// TIA Portal V17 export
// export: Created 2025-03-07T09:18:31.7382739Z, ExportSetting WithDefaults, DisplayName Totally Integrated Automation Portal, DisplayVersion V17 Update 8, DisplayName TIA Portal Openness, DisplayVersion V17 Update 8, DisplayName TIA Portal Version Control Interface, DisplayVersion V17, DisplayName SINAMICS Startdrive Advanced, DisplayVersion V17 SP2, DisplayName SINAMICS Startdrive G110M, G120, G120C, G120D, G120P, G115D, DisplayVersion V17 SP2, DisplayName SINAMICS Startdrive G130, G150, S120, S150, SINAMICS MV, S210, DisplayVersion V17 SP2, DisplayName STEP 7 Professional, DisplayVersion V17 Update 8, DisplayName SINUMERIK ONE STEP 7 Toolbox, DisplayVersion V17 Update 12, DisplayName SINUMERIK 840D sl STEP 7 Toolbox, DisplayVersion V17 Update 12, DisplayName STEP 7 Safety, DisplayVersion V17 Update 6, DisplayName WinCC Advanced, DisplayVersion V17 Update 8
DATA_BLOCK "LTLP_OperatingModeData"   // DB547
{ S7_Optimized_Access := 'FALSE'; DB_Accessible_From_OPC_UA := 'FALSE' }
VERSION : 0.1
// stored: AutoNumber true, DBAccessibleFromOPCUA false, DBAccessibleFromWebserver true, InstanceOfName LTLP_typeOperatingMode, InstanceOfType UDT, IsOnlyStoredInLoadMemory false, IsWriteProtectedInAS false
"LTLP_typeOperatingMode"
   // VAR RETAIN
   //    automaticMode : Struct
   //       tlFunctionAutomaticMode { S7_SetPoint := 'True'} : "LTLP_typeEnableFucntions";
   //       tlFunctionSingleMode { S7_SetPoint := 'True'} : "LTLP_typeEnableFucntions";
   //       tlFunctionSingleStepMode { S7_SetPoint := 'True'} : "LTLP_typeEnableFucntions";
   //       tlFunctionSetupMode { S7_SetPoint := 'True'} : "LTLP_typeEnableFucntions";
   //    END_STRUCT;
   //    setupMode : Struct
   //       tlFunctionSetupMode { S7_SetPoint := 'True'} : "LTLP_typeEnableFucntions";
   //    END_STRUCT;
   //    processMonitoring : Struct
   //       tlFunctionSingleMode { S7_SetPoint := 'True'} : "LTLP_typeEnableFucntions";
   //       tlFunctionSingleStep { S7_SetPoint := 'True'} : "LTLP_typeEnableFucntions";
   //    END_STRUCT;
   //    specialOperatingMode : Struct
   //       tlFunctionAutomaticMode { S7_SetPoint := 'True'} : "LTLP_typeEnableFucntions";
   //       tlFunctionSingleMode { S7_SetPoint := 'True'} : "LTLP_typeEnableFucntions";
   //    END_STRUCT;
   //    dataStorage : Struct
   //       posTriggerAutomaticMode : Bool;
   //       posTriggerSetupMode : Bool;
   //       posTriggerProcessMonitoring : Bool;
   //       posTriggerSpecialOperationMode : Bool;
   //       reserve14 : Bool;
   //       reserve15 : Bool;
   //       reserve16 : Bool;
   //       reserve17 : Bool;
   //       tlFunctionAutomaticMode : Bool;
   //       tlFunctionSingleMode : Bool;
   //       tlFunctionSingleStep : Bool;
   //       tlFunctionSetupMode : Bool;
   //    END_STRUCT;
   // END_VAR
BEGIN
END_DATA_BLOCK
